{attribute 'qualified_only'}
{attribute 'strict'}
TYPE EFeedbackMsgMicroEpsilonDistanceSensor :
(
	StateMsg := 1,
	StatusMsg := 2,
	IsAliveMsg := 3,
	DistanceMsg := 10,
	IdMsg,
	CustomMsg
);
END_TYPE

(* stored: Version 1.1.0.1, ProductVersion 3.1.4024.12
   DUT EFeedbackMsgMicroEpsilonDistanceSensor: Id {84a9f530-6117-46c2-afe2-41c743e97e9d} *)
